Staubli VAL3: AllMotion.pgx

public program AllMotion(string x_sPrd)
  local bool l_bRes
  local num l_ni
  local num l_nSize
begin
  //
  //判断安全位置
  call chkAtHome(l_bRes)
  if !l_bRes
    return
  endIf
  //
  PublicData:sStatus="stop"
  //正在加工的路径
  if PublicData:sCurrentPrd!=x_sPrd
    PublicData:sCurrentPrd=x_sPrd
    l_ni=0
    while l_ni<size(sProductList) and find(sProductList[l_ni],"P")<0
      l_ni=l_ni+1
    endWhile
    //初始化计数
    l_nSize=l_ni
    resize(PublicData:nCompenCount,1,l_nSize)
    for l_ni=0 to l_nSize-1
      PublicData:nCompenCount[l_ni]=0
    endFor
  endIf
  //
  taskCreate "control",100,Control()
  taskCreate "motion",100,WholeMotion(x_sPrd)
  call MotionPage()
end
